PROGRAM InitTCPIP
VAR
	sSrvNetID 		: T_AmsNetID := '';(* TwinCAT TCP/IP server network address *)
	fbCloseAll		: FB_SocketCloseAll;
END_VAR

(* On PLC reset or program download close all created/opened sockets/connections *)
fbCloseAll( sSrvNetID := sSrvNetID, bExecute:= bInitTCPIP );
IF fbCloseAll.bBusy OR fbCloseAll.bError THEN
	RETURN;
END_IF
bInitTCPIP := FALSE;

END_PROGRAM

(* stored: Version 1.1.0.1, ProductVersion 3.1.4024.11
   POU InitTCPIP: Id {1ab60bce-2155-45d7-b4bb-787adb64acf0}, SpecialFunc None *)
